{attribute addProperty BoxType "EL4732-0001-0000"}
{attribute addProperty Id "Cycle_CounterAT %Q*Cycle_Counter_485675001620Sample_0AT %Q*Sample_6DB94BDA3240WcStateAT %I*WcState_64F6A8C6810InfoDataAT %I*InfoData_7231B2DD80100"}
{attribute addProperty CRC "1430642600"}
{attribute addProperty SizeInBites "136"}
{attribute addProperty SizeInBytes "17"}
TYPE EL4732_13EEB3C3 :
STRUCT
	{attribute addProperty Name "Cycle_Counter"}
	Cycle_Counter : Cycle_Counter_48567500;
	{attribute addProperty Name "Sample_0"}
	Sample_0 : Sample_6DB94BDA;
	{attribute addProperty Name "WcState"}
	WcState : WcState_64F6A8C6;
	{attribute addProperty Name "InfoData"}
	InfoData : InfoData_7231B2DD;
END_STRUCT
END_TYPE

(* stored: Version 1.2.0.0, ProductVersion 3.1.4024.9
   DUT EL4732_13EEB3C3: Id {54f94510-28e6-4aa8-b067-955b1d83c82d} *)
